Fanuc KAREL source: KT00187.KL

PROGRAM KT00187
%NOLOCKGROUP
VAR
  H1: ARRAY[2] OF SHORT
  R2: REAL
  OUT: INTEGER
BEGIN
  H1[1] = 2
    R2 = 3.0
  OUT = H1[1] MOD R2
END KT00187
